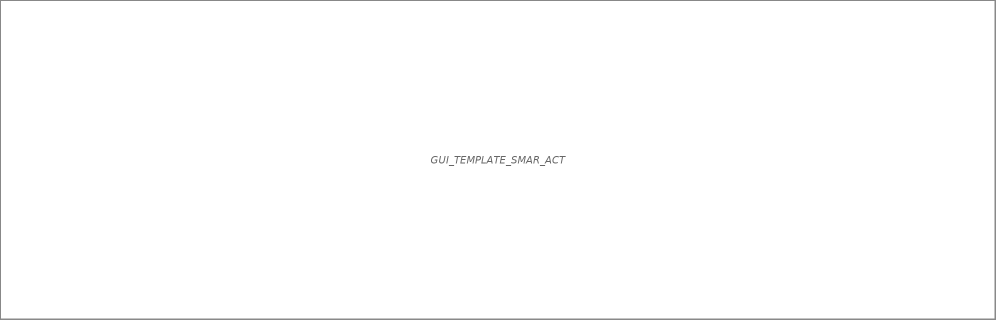
VISUALIZATION GUI_SmarAct_SIM  // 996x320
    Frame (0,0 996x320)
        shows GUI_TEMPLATE_SMAR_ACT(m_Instance := MAIN.SmarAct_Sim)
END_VISUALIZATION

(* stored: Version 1.1.0.1, ProductVersion 3.1.4024.10
   Visu GUI_SmarAct_SIM: Id {3335fea1-9839-407d-9788-cfcb0bf1f6aa} *)
